# EPICS substitutions: elioApp/Db/EL2798.substitutions
file EL2798.template { pattern
{ CHAN	}
{ 1	}
{ 2	}
{ 3	}
{ 4	}
{ 5	}
{ 6	}
{ 7	}
{ 8	}
}
